% RSLogix 500 project P3_INVENTORY_MANAGEMENT.RSS, saved by version 8.30.00.16 %
PROJECT "BARCODE"    % processor: Bul.1763 MicroLogix 1100 Series B %

PROGRAM FILES
  LAD 2 "MAIN"  7 rungs
  LAD 3 "JUNKYARD"  1 rungs  % JUNKYARD %

DATA FILES
  O0 OUTPUT  4 elements
  I1 INPUT  6 elements
  S2 STATUS  66 elements
  B3 BINARY  1 elements
  T4 TIMER  1 elements
  C5 COUNTER  1 elements
  R6 CONTROL  1 elements
  N7 INTEGER  6 elements
  F8 FLOAT  1 elements
  ST9 STRING  13 elements

LADDER 2 "MAIN"
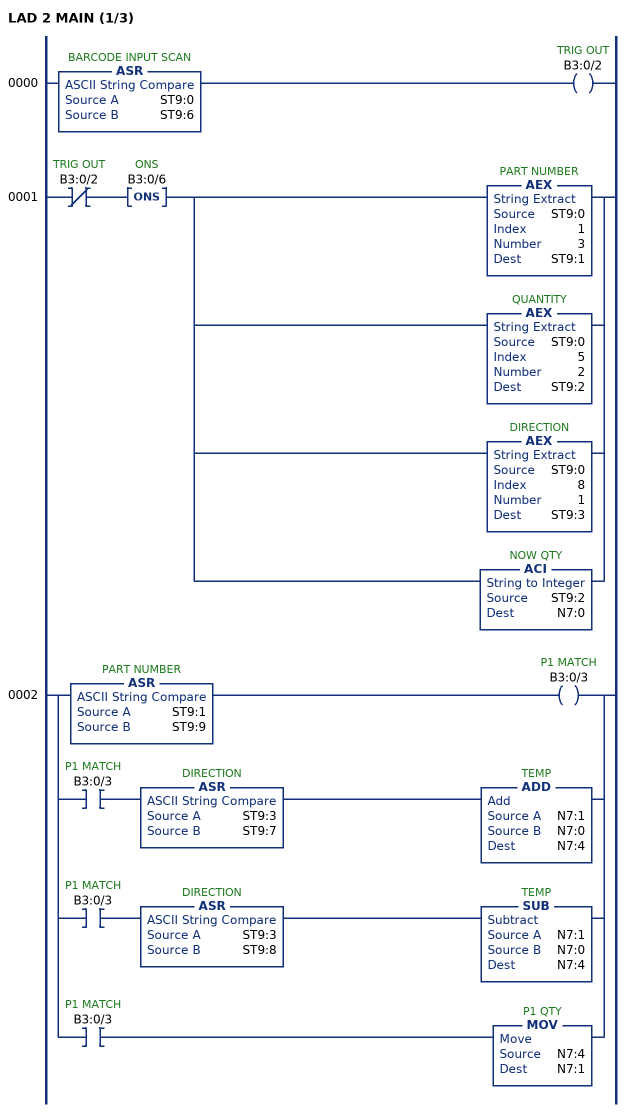
% Rung: 0 %
SOR ASR ST9:0 ST9:6 OTE B3:0/2 EOR
%   ST9:0  "BARCODE INPUT SCAN" %
%   B3:0/2  "TRIG OUT" %
% Rung: 1 %
SOR XIO B3:0/2 ONS B3:0/6 BST AEX ST9:0 1 3 ST9:1 NXB AEX ST9:0 5 2 ST9:2 NXB AEX ST9:0 8 1 ST9:3 NXB ACI ST9:2 N7:0 BND EOR
%   B3:0/2  "TRIG OUT" %
%   B3:0/6  "ONS" %
%   ST9:0  "BARCODE INPUT SCAN" %
%   ST9:1  "PART NUMBER" %
%   ST9:2  "QUANTITY" %
%   ST9:3  "DIRECTION" %
%   N7:0  "NOW QTY" %
% Rung: 2 %
SOR BST ASR ST9:1 ST9:9 OTE B3:0/3 NXB XIC B3:0/3 ASR ST9:3 ST9:7 ADD N7:1 N7:0 N7:4 NXB XIC B3:0/3 ASR ST9:3 ST9:8 SUB N7:1 N7:0 N7:4 NXB XIC B3:0/3 MOV N7:4 N7:1 BND EOR
%   ST9:1  "PART NUMBER" %
%   ST9:9  "PRODUCT 1 PART NO" %
%   B3:0/3  "P1 MATCH" %
%   ST9:3  "DIRECTION" %
%   ST9:7  "INWARD" %
%   N7:1  "P1 QTY" %
%   N7:0  "NOW QTY" %
%   N7:4  "TEMP" %
%   ST9:8  "OUTWARD" %

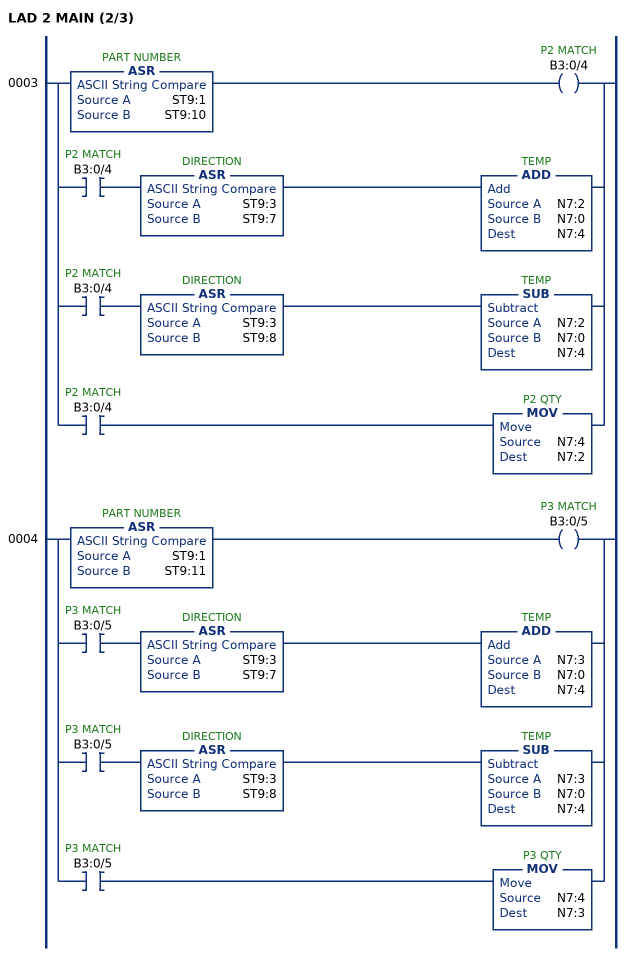
% Rung: 3 %
SOR BST ASR ST9:1 ST9:10 OTE B3:0/4 NXB XIC B3:0/4 ASR ST9:3 ST9:7 ADD N7:2 N7:0 N7:4 NXB XIC B3:0/4 ASR ST9:3 ST9:8 SUB N7:2 N7:0 N7:4 NXB XIC B3:0/4 MOV N7:4 N7:2 BND EOR
%   ST9:1  "PART NUMBER" %
%   ST9:10  "PRODUCT 2 PART NO" %
%   B3:0/4  "P2 MATCH" %
%   ST9:3  "DIRECTION" %
%   ST9:7  "INWARD" %
%   N7:2  "P2 QTY" %
%   N7:0  "NOW QTY" %
%   N7:4  "TEMP" %
%   ST9:8  "OUTWARD" %
% Rung: 4 %
SOR BST ASR ST9:1 ST9:11 OTE B3:0/5 NXB XIC B3:0/5 ASR ST9:3 ST9:7 ADD N7:3 N7:0 N7:4 NXB XIC B3:0/5 ASR ST9:3 ST9:8 SUB N7:3 N7:0 N7:4 NXB XIC B3:0/5 MOV N7:4 N7:3 BND EOR
%   ST9:1  "PART NUMBER" %
%   ST9:11  "PRODUCT 3 PART NO" %
%   B3:0/5  "P3 MATCH" %
%   ST9:3  "DIRECTION" %
%   ST9:7  "INWARD" %
%   N7:3  "P3 QTY" %
%   N7:0  "NOW QTY" %
%   N7:4  "TEMP" %
%   ST9:8  "OUTWARD" %

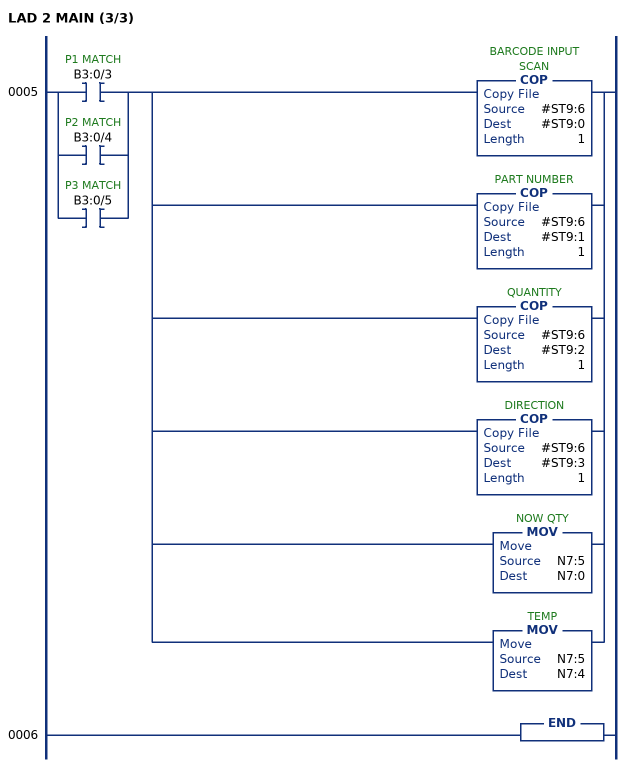
% Rung: 5 %
SOR BST XIC B3:0/3 NXB XIC B3:0/4 NXB XIC B3:0/5 BND BST COP #ST9:6 #ST9:0 1 NXB COP #ST9:6 #ST9:1 1 NXB COP #ST9:6 #ST9:2 1 NXB COP #ST9:6 #ST9:3 1 NXB MOV N7:5 N7:0 NXB MOV N7:5 N7:4 BND EOR
%   B3:0/3  "P1 MATCH" %
%   B3:0/4  "P2 MATCH" %
%   B3:0/5  "P3 MATCH" %
%   ST9:0  "BARCODE INPUT SCAN" %
%   ST9:1  "PART NUMBER" %
%   ST9:2  "QUANTITY" %
%   ST9:3  "DIRECTION" %
%   N7:5  "ZERO" %
%   N7:0  "NOW QTY" %
%   N7:4  "TEMP" %
% Rung: 6 %
SOR END EOR

OTHER DOCUMENTED ADDRESSES
  B3:0/0  "SCAN TRIG"
  B3:0/1  "SCAN ONS"
  C5:0/DN  "CTR DN"
  ST9:4  "EMPTY STRING"

DATA TABLE (non-zero values as saved)
DATA B3
% B3:0 % 0X0007
DATA C5
% .PRE .ACC %
% C5:0 % 1 0
DATA ST9
% ST9:7 % "1"
% ST9:8 % "2"
% ST9:9 % "123"
% ST9:10 % "456"
% ST9:11 % "789"
